# EPICS substitutions: CsHeaterApp/Db/Watlow_PM_Limits.substitutions
####Macro Definitions####

#### Global ####
# (ta)	- Target Area
# (ss)	- Device Name
# (ch)	- Channel

file Watlow_PM_Limits.template
{
pattern	{       ta,          ss, Ain}
        {SP_Cesium, Oven_Heater,   0}
}
